FUNCTION_BLOCK StringBuilder
VAR
	result : STRING(1000);
END_VAR

METHOD concatStringArray : STRING(1000)
VAR_IN_OUT
	arr : ARRAY[*] OF STRING;
END_VAR
VAR
	temp : STRING(1000);
END_VAR
END_METHOD

METHOD concatWith : REFERENCE TO StringBuilder
VAR_INPUT
	target : STRING;
END_VAR
CONCAT2(ADR(result), ADR(target), ADR(result), SIZEOF(result));
concatWith REF= THIS^;
END_METHOD

METHOD getResult : STRING(1000)
getResult := result;
END_METHOD

METHOD reset : BOOL
VAR_INPUT
END_VAR
result := '';
END_METHOD

END_FUNCTION_BLOCK

(* stored: Version 1.1.0.1, ProductVersion 3.1.4024.11
   POU StringBuilder: Id {22f9fe77-0400-479d-89ca-12725f28136a}, SpecialFunc None
   Method concatStringArray: Id {6d4d58b1-72e5-4e1d-aedb-b37876c0d39b}
   Method concatWith: Id {ad17e71b-95ca-4f38-a153-4c45f5f8fd3c}
   Method getResult: Id {27cff9f3-46ca-49f6-be7b-07517171a027}
   Method reset: Id {c2e2ebfe-dcac-45ca-9376-8551eeb7ba0d} *)
